Staubli VAL3: getSizeAction.pgx

public program getSizeAction(num& x_nSize)
begin
  // mutex it
  setMutex(bActionMutex)
  // give back the action on first element
  x_nSize=size(aAction)
  //release
  bActionMutex=false
end
